(* PLC project SafeLOGIC-1, BrAutomation SafeDESIGNER  4.3.3.7 *)
(* stored: companyURL http://www.br-automation.com, creationDateTime Tue Jun 23 09:46:05 2020 *)

PROGRAM SafeModules_OK

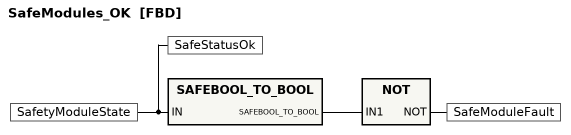
(* FBD diagram, written out as Structured Text *)
SafeStatusOk := SafetyModuleState;
SafeModuleFault := NOT SAFEBOOL_TO_BOOL(SafetyModuleState);
END_PROGRAM
